FUNCTION_BLOCK FB_ShowControlPanel
VAR_INPUT
	arrSwitch		: ARRAY[1..C_MAXCOMMANDS] OF BOOL;
END_VAR
VAR
	aiCommand		: ARRAY[1..C_MAXCOMMANDS] OF I_Command;	
	arrRtrig		: ARRAY[1..C_MAXCOMMANDS] OF R_TRIG;
	nIndex			: INT;
END_VAR
VAR CONSTANT
	C_MAXCOMMANDS	: INT := 12;
END_VAR

FOR nIndex := 1 TO C_MAXCOMMANDS DO
	arrRtrig[nIndex](CLK := arrSwitch[nIndex]);
	IF aiCommand[nIndex] <> 0 THEN
		
		IF arrRtrig[nIndex].Q AND (aiCommand[nIndex] <> 0)THEN
				aiCommand[nIndex].Execute();	
		END_IF
				
	END_IF
END_FOR

METHOD FB_init : BOOL
VAR_INPUT
	bInitRetains : BOOL; // if TRUE, the retain variables are initialized (warm start / cold start)
	bInCopyCode : BOOL;  // if TRUE, the instance afterwards gets moved into the copy code (online change)
END_VAR
VAR
	nIndex : INT;
END_VAR
FOR nIndex := 1 TO C_MAXCOMMANDS DO
	aiCommand[nIndex] := 0;
END_FOR
END_METHOD

METHOD SetCommand : BOOL
VAR_INPUT
	nPosition		: INT;
	iCommand		: I_Command;
END_VAR
IF ((nPosition >= 1) AND (nPosition <= C_MAXCOMMANDS) AND (iCommand <> 0)) THEN
		THIS^.aiCommand[nPosition] := iCommand;
END_IF
END_METHOD

END_FUNCTION_BLOCK

(* stored: Version 1.1.0.1, ProductVersion 3.1.4022.18
   POU FB_ShowControlPanel: Id {856921ab-341a-4bf4-ae97-d8ce6d9d2448}, SpecialFunc None
   Method FB_init: Id {69122625-f844-40eb-802f-24c07b744651}
   Method SetCommand: Id {7957bb33-29b3-4bd2-a13e-9fd2457c016f} *)
